INTERFACE I_AnyBufferStrategy

METHOD Clear : BOOL
END_METHOD

PROPERTY isEmpty : BOOL
GET
END_GET
END_PROPERTY

PROPERTY isFull : BOOL
GET
END_GET
END_PROPERTY

END_INTERFACE

(* stored: Version 1.1.0.1, ProductVersion 3.1.4026.18
   Itf I_AnyBufferStrategy: Id {f5ddd2a6-d5a1-465f-9d4c-2073f3f17d30}
   Method Clear: Id {7cbbf9fc-5ef5-4ab4-90ba-2b494932ede4}
   Property isEmpty: Id {ee0be38f-0fe9-4e01-9dce-e3504330ac64}
   Get Get: Id {ac0f001e-e3b6-4cd3-a991-3164a019a046}
   Property isFull: Id {25f592d5-1274-42f1-a8e2-81bb2c82d30c}
   Get Get: Id {d101225f-6f55-431c-a488-732b8a685df2} *)
